// TIA Portal V16 export
// export: Created 2025-05-30T16:36:22.7111105Z, ExportSetting WithDefaults, DisplayName Totally Integrated Automation Portal, DisplayVersion V16, DisplayName TIA Portal Version Control Interface, DisplayVersion V16, DisplayName TIA Portal Openness, DisplayVersion V16, DisplayName STEP 7 Professional, DisplayVersion V16, DisplayName STEP 7 Safety, DisplayVersion V16, DisplayName WinCC Advanced, DisplayVersion V16
DATA_BLOCK "ESB_Lamp_Block"   // DB34
VERSION : 0.1
// stored: AutoNumber true, InstanceOfName ESB_Flash_Warning_Block, InstanceOfType FB
"ESB_Flash_Warning_Block"
   // VAR_INPUT
   //    "Safety Feedback Contact" : Bool;
   //    "WarningTimer Time 1" : Time;
   //    "WarningTimer Time 2" : Time;
   // END_VAR
   // VAR_OUTPUT
   //    "Warning Ouput Contact" : Bool;
   //    "ET WarningTimer 1" : Time;
   //    "ET WarningTimer 2" : Time;
   // END_VAR
BEGIN
END_DATA_BLOCK
